% RSLogix 500 project conveyor belts.RSS, saved by version 8.30.00.16 %
PROJECT "UNTITLED"    % processor: Bul.1763 MicroLogix 1100 Series B %

PROGRAM FILES
  LAD 2 "MAIN"  4 rungs
  LAD 3 "INPUT"  5 rungs
  LAD 4 "OUTPUT"  4 rungs
  LAD 5 "CONTROL"  13 rungs

DATA FILES
  O0 OUTPUT  4 elements
  I1 INPUT  6 elements
  S2 STATUS  66 elements
  B3 BINARY  2 elements
  T4 TIMER  4 elements
  C5 COUNTER  1 elements
  R6 CONTROL  1 elements
  N7 INTEGER  1 elements
  F8 FLOAT  1 elements

LADDER 2 "MAIN"
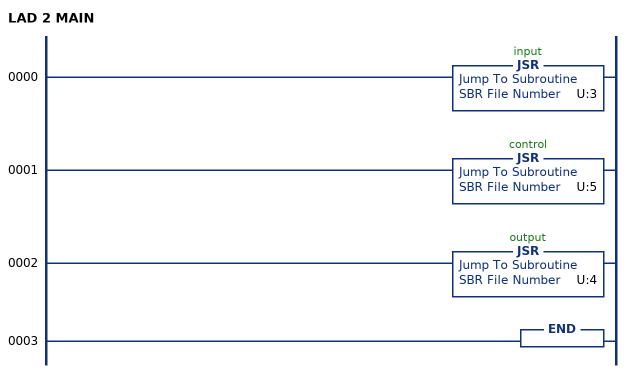
% Rung: 0 %
SOR JSR U:3 EOR
%   U:3  "input" %
% Rung: 1 %
SOR JSR U:5 EOR
%   U:5  "control" %
% Rung: 2 %
SOR JSR U:4 EOR
%   U:4  "output" %
% Rung: 3 %
SOR END EOR

LADDER 3 "INPUT"
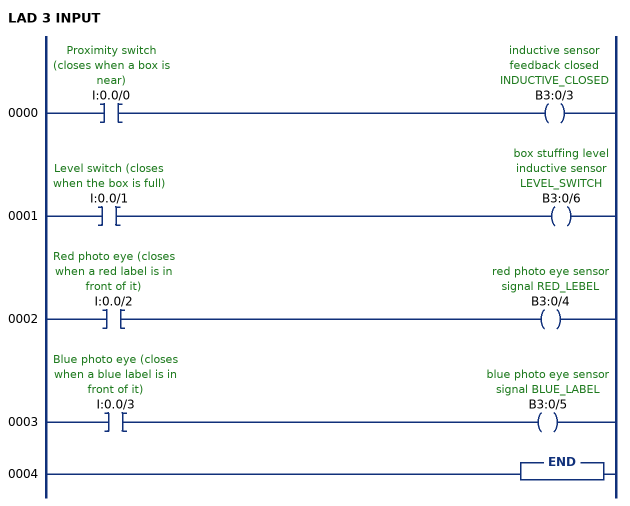
% Rung: 0 %
SOR XIC I:0.0/0 OTE B3:0/3 EOR
%   I:0.0/0  "Proximity switch (closes when a box is near)" %
%   B3:0/3  INDUCTIVE_CLOSED  "inductive sensor feedback closed" %
% Rung: 1 %
SOR XIC I:0.0/1 OTE B3:0/6 EOR
%   I:0.0/1  "Level switch (closes when the box is full)" %
%   B3:0/6  LEVEL_SWITCH  "box stuffing level inductive sensor" %
% Rung: 2 %
SOR XIC I:0.0/2 OTE B3:0/4 EOR
%   I:0.0/2  "Red photo eye (closes when a red label is in front of it)" %
%   B3:0/4  RED_LEBEL  "red photo eye sensor signal" %
% Rung: 3 %
SOR XIC I:0.0/3 OTE B3:0/5 EOR
%   I:0.0/3  "Blue photo eye (closes when a blue label is in front of it)" %
%   B3:0/5  BLUE_LABEL  "blue photo eye sensor signal" %
% Rung: 4 %
SOR END EOR

LADDER 4 "OUTPUT"
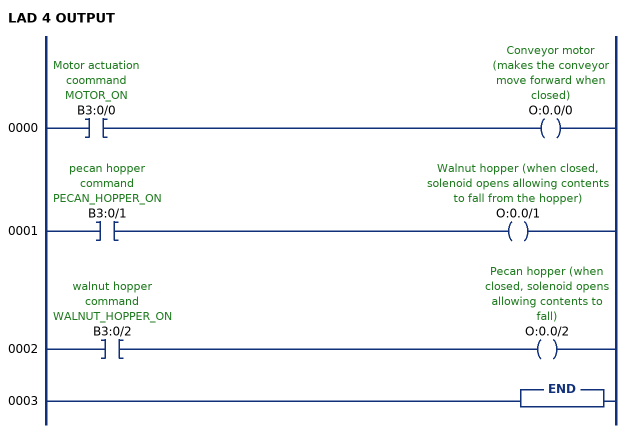
% Rung: 0 %
SOR XIC B3:0/0 OTE O:0.0/0 EOR
%   B3:0/0  MOTOR_ON  "Motor actuation coommand" %
%   O:0.0/0  "Conveyor motor (makes the conveyor move forward when closed)" %
% Rung: 1 %
SOR XIC B3:0/1 OTE O:0.0/1 EOR
%   B3:0/1  PECAN_HOPPER_ON  "pecan hopper command" %
%   O:0.0/1  "Walnut hopper (when closed, solenoid opens allowing contents to fall from the hopper)" %
% Rung: 2 %
SOR XIC B3:0/2 OTE O:0.0/2 EOR
%   B3:0/2  WALNUT_HOPPER_ON  "walnut hopper command" %
%   O:0.0/2  "Pecan hopper (when closed, solenoid opens allowing contents to fall)" %
% Rung: 3 %
SOR END EOR

LADDER 5 "CONTROL"
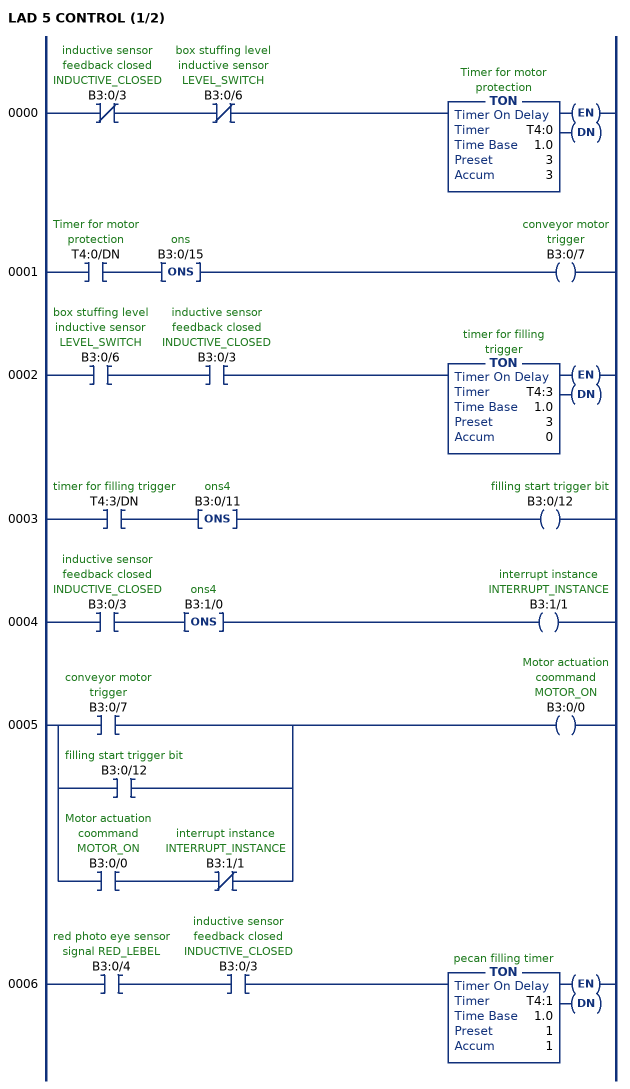
% Rung: 0 %
SOR XIO B3:0/3 XIO B3:0/6 TON T4:0 1.0 3 3 EOR
%   B3:0/3  INDUCTIVE_CLOSED  "inductive sensor feedback closed" %
%   B3:0/6  LEVEL_SWITCH  "box stuffing level inductive sensor" %
%   T4:0  "Timer for motor protection" %
% Rung: 1 %
SOR XIC T4:0/DN ONS B3:0/15 OTE B3:0/7 EOR
%   T4:0  "Timer for motor protection" %
%   B3:0/15  "ons" %
%   B3:0/7  "conveyor motor trigger" %
% Rung: 2 %
SOR XIC B3:0/6 XIC B3:0/3 TON T4:3 1.0 3 0 EOR
%   B3:0/6  LEVEL_SWITCH  "box stuffing level inductive sensor" %
%   B3:0/3  INDUCTIVE_CLOSED  "inductive sensor feedback closed" %
%   T4:3  "timer for filling trigger" %
% Rung: 3 %
SOR XIC T4:3/DN ONS B3:0/11 OTE B3:0/12 EOR
%   T4:3  "timer for filling trigger" %
%   B3:0/11  "ons4" %
%   B3:0/12  "filling start trigger bit" %
% Rung: 4 %
SOR XIC B3:0/3 ONS B3:1/0 OTE B3:1/1 EOR
%   B3:0/3  INDUCTIVE_CLOSED  "inductive sensor feedback closed" %
%   B3:1/0  "ons4" %
%   B3:1/1  INTERRUPT_INSTANCE  "interrupt instance" %
% Rung: 5 %
SOR BST BST XIC B3:0/7 NXB XIC B3:0/12 BND NXB XIC B3:0/0 XIO B3:1/1 BND OTE B3:0/0 EOR
%   B3:0/7  "conveyor motor trigger" %
%   B3:0/12  "filling start trigger bit" %
%   B3:0/0  MOTOR_ON  "Motor actuation coommand" %
%   B3:1/1  INTERRUPT_INSTANCE  "interrupt instance" %
% Rung: 6 %
SOR XIC B3:0/4 XIC B3:0/3 TON T4:1 1.0 1 1 EOR
%   B3:0/4  RED_LEBEL  "red photo eye sensor signal" %
%   B3:0/3  INDUCTIVE_CLOSED  "inductive sensor feedback closed" %
%   T4:1  "pecan filling timer" %

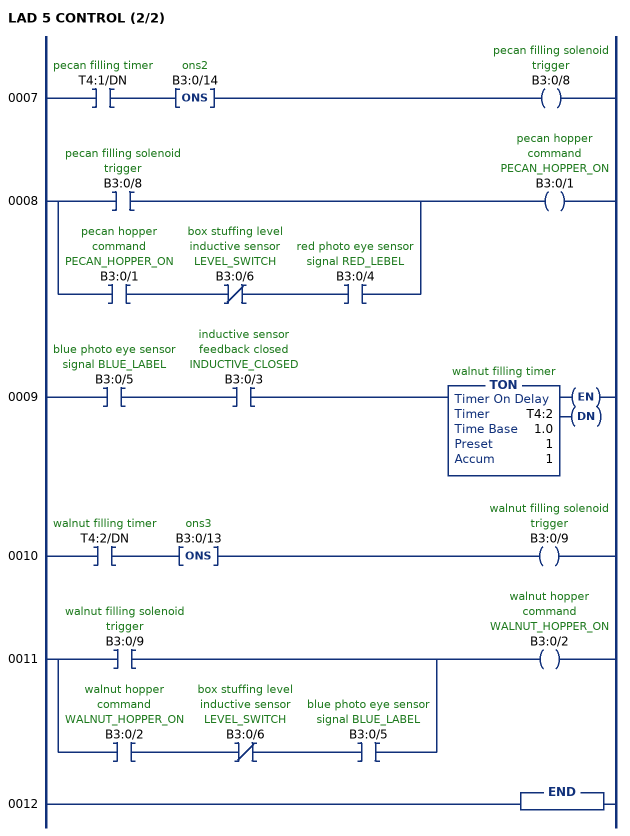
% Rung: 7 %
SOR XIC T4:1/DN ONS B3:0/14 OTE B3:0/8 EOR
%   T4:1  "pecan filling timer" %
%   B3:0/14  "ons2" %
%   B3:0/8  "pecan filling solenoid trigger" %
% Rung: 8 %
SOR BST XIC B3:0/8 NXB XIC B3:0/1 XIO B3:0/6 XIC B3:0/4 BND OTE B3:0/1 EOR
%   B3:0/8  "pecan filling solenoid trigger" %
%   B3:0/1  PECAN_HOPPER_ON  "pecan hopper command" %
%   B3:0/6  LEVEL_SWITCH  "box stuffing level inductive sensor" %
%   B3:0/4  RED_LEBEL  "red photo eye sensor signal" %
% Rung: 9 %
SOR XIC B3:0/5 XIC B3:0/3 TON T4:2 1.0 1 1 EOR
%   B3:0/5  BLUE_LABEL  "blue photo eye sensor signal" %
%   B3:0/3  INDUCTIVE_CLOSED  "inductive sensor feedback closed" %
%   T4:2  "walnut filling timer" %
% Rung: 10 %
SOR XIC T4:2/DN ONS B3:0/13 OTE B3:0/9 EOR
%   T4:2  "walnut filling timer" %
%   B3:0/13  "ons3" %
%   B3:0/9  "walnut filling solenoid trigger" %
% Rung: 11 %
SOR BST XIC B3:0/9 NXB XIC B3:0/2 XIO B3:0/6 XIC B3:0/5 BND OTE B3:0/2 EOR
%   B3:0/9  "walnut filling solenoid trigger" %
%   B3:0/2  WALNUT_HOPPER_ON  "walnut hopper command" %
%   B3:0/6  LEVEL_SWITCH  "box stuffing level inductive sensor" %
%   B3:0/5  BLUE_LABEL  "blue photo eye sensor signal" %
% Rung: 12 %
SOR END EOR

OTHER DOCUMENTED ADDRESSES
  B3:0/10  AFTER_FILLING_BIT  "after filling start bit"

DATA TABLE (non-zero values as saved)
DATA B3
% B3:0 % 0XE037 0X0000
DATA T4
% .PRE .ACC %
% T4:0 % 3 3
% T4:1 % 1 1
% T4:2 % 1 1
% T4:3 % 3 0
